// TIA Portal V20 export
// export: Created 2025-12-01T14:57:08.1261523Z, ExportSetting None, DisplayName Totally Integrated Automation Portal, DisplayVersion V20 Update 3, DisplayName TIA Portal Openness, DisplayVersion V20 Update 3, DisplayName TIA Portal Version Control Interface, DisplayVersion V20 Update 3, DisplayName STEP 7 Professional, DisplayVersion V20 Update 3, DisplayName STEP 7 Safety, DisplayVersion V20 Update 2, DisplayName WinCC Basic/Comfort/Advanced, DisplayVersion V20 Update 3, DisplayName WinCC Professional, DisplayVersion V20 Update 3, DisplayName WinCC Unified, DisplayVersion V20 Update 3
FUNCTION "FC861_Informe_DispositivoMesa" : Void   // FC861, STL
{ S7_Optimized_Access := 'FALSE' }
// stored: AutoNumber false
   VAR_INPUT
      Mesa : UInt;
   END_VAR
   VAR_OUTPUT
      Informe_DispositivoMesa : "UDT_Informe_DispositivoMesa";
   END_VAR
   VAR_TEMP
      Relleno : Byte;
      ValorReturn : Int;
   END_VAR
BEGIN

NETWORK
TITLE = Inicializar
//////////////////////////////////////////////////////////////////////
/// Inicializar Variables

      L     0;
      T     #Relleno;

      CALL  FILL
      ( BVAL    := #Relleno,
        RET_VAL := #ValorReturn,
        BLK     := #Informe_DispositivoMesa
      );



NETWORK
TITLE = Crear Informe
//////////////////////////////////////////////////////////////////////
/// Crear Informe del Dispositivo

      SET;
      A     "DB831_Mesas".Mesas[#Mesa].Memorias.DesHabilitado;
      =     #Informe_DispositivoMesa.Bits.DesHabilitado;

      SET;
      AN    "DB831_Mesas".Mesas[#Mesa].Memorias.DesHabilitado;
      =     #Informe_DispositivoMesa.Bits.Habilitado;


//////////////////////////////////////////////////////////////////////
/// Calculo de Prioridad

      L     "DB831_Mesas".Mesas[#Mesa].Prioridad;
      T     #Informe_DispositivoMesa.Prioridad;
      BE;  // - Finalizar bloque

END_FUNCTION
